TYPE ST_Simplex_Halt :
STRUCT
	nMotorFluxVoltage : INT;
END_STRUCT
END_TYPE

(* stored: Version 1.1.0.1, ProductVersion 3.1.4020.12
   DUT ST_Simplex_Halt: Id {1deddee4-1d00-4b74-9a1d-956eedfbd1b4} *)
